// TwinCAT 3 PLC project CounterToOutput
// ProgramVersion: 3.1.0.8
// libraries:
//   VisuElem3DPath, 3.5.6.0 (System)
//   VisuElemMeter, 3.5.6.0 (System)
//   VisuElems, 3.5.6.10 (System)
//   VisuElemsDateTime, 3.5.6.0 (System)
//   VisuElemsSpecialControls, 3.5.6.0 (System)
//   VisuElemsWinControls, 3.5.6.0 (System)
//   VisuElemTextEditor, 3.5.6.0 (System)
//   visuinputs, 3.5.6.0 (system)
//   VisuNativeControl, 3.5.6.0 (System)
//   Tc2_ModbusSrv, * (Beckhoff Automation GmbH)
//   Tc2_Standard, * (Beckhoff Automation GmbH)
//   Tc2_System, * (Beckhoff Automation GmbH)
//   Tc3_Interfaces, * (Beckhoff Automation GmbH)
//   Tc3_Module, * (Beckhoff Automation GmbH)
// project tree:
//   / GlobalTextList.TcGTLO, Visualization Manager.TcVMO (not stored)
//   GVLs/ G_IO.TcGVL
//   POUs/ stMain.TcPOU
// real-time tasks:
//   TASK PlcTask: cycle T#10ms, priority 20, ADS port 350
// I/O:
//   DEVICE Device 1 (EtherCAT), AmsNetId 5.20.215.224.2.1
//     Term 1 (EK1200) [EK1200-5000 EtherCAT Power supply (2A E-Bus)]
//       Term 2 (EL3058) [EL3058 8Ch. Ana. Input 4-20mA]
//       Term 3 (EL4028) [EL4028 8Ch. Ana. Output 4-20mA, 12bit]
//       Term 4 (EL1808) [EL1808 8Ch. Dig. Input 24V, 3ms]
//       Term 5 (EL2808) [EL2808 8Ch. Dig. Output 24V, 0.5A]
//       Term 6 (EL3068) [EL3068 8Ch. Ana. Input 0-10V]
//       Term 7 (EL4008) [EL4008 8Ch. Ana. Output 0-10V, 12bit]
//       Term 8 (EL9011) [EL9011 End Terminal]

// ---- GVLs/G_IO.TcGVL
VAR_GLOBAL
	
	AOUT AT %Q*	:	ARRAY[1..2] OF INT;
	
	XMEAS:	ARRAY[1..41] OF LREAL;
	MBS_XMEAS:	ARRAY[1..2] OF REAL;
	
END_VAR

// ---- POUs/stMain.TcPOU
PROGRAM stMain	
VAR

	OUT_VAL:	REAL := 0;	
	
	T1:	TON;
END_VAR


T1(IN:=(T1.Q=FALSE),PT:=T#1.0S,);

IF T1.Q THEN

	AOUT[1]		:= REAL_TO_INT(OUT_VAL);
	AOUT[2]		:= REAL_TO_INT(4*OUT_VAL);
	
	OUT_VAL := OUT_VAL + 100.0;
	
	IF (OUT_VAL > 32768.0/8.0) THEN
		OUT_VAL := 0;
	END_IF
	
END_IF

END_PROGRAM
